PROGRAM MAIN
VAR
END_VAR

END_PROGRAM

(* stored: Version 1.1.0.1
   POU MAIN: Id {ceb1e854-a12e-4d2e-97cf-4377a49f0fe3} *)
